(* CODESYS project wago_aws_iot_example_v0.2.01.ecp

Project tree, tasks and I/O mapping:
  PFC200_CS_2ETH_RS : 750-8202 PFC200 2ETH RS, WAGO, order no. 0750-8202, version 5.11.1.16
    application Application
      libraries: 
      task PLC_Task (cyclic, interval t#10ms, priority 14) calls PLC_PRG
      task VISU_TASK (cyclic, interval 100 ms, priority 15) calls VisuElems.Visu_Prg
      visualisation Visualization
      function block UPDATE_AWS_IOT_THING_SHADOW [ST]: PUB_STRING
      program PLC_PRG [ST]
      visualisation Shadow_Attribute_Visu
      image pool ImagePool
      function block GET_AWS_IOT_THING_SHADOW [ST]: CURL_STRING
      function funC_TO_F [ST]
    DeviceAdapter
    Kbus : Kbus, WAGO, version 1.4.0.2
        unmapped channels: K-BUS diagnostics
      _4_AI_4_20mA_s_e_1 : 0750-0455, WAGO, order no. 0750-0455, version 0.0.0.12
          settings: K-BUS Module slot index = 1
          unmapped channels: _IW 1, _IW 2, _IW 3, _IW 4
        DeviceAdapter
      _2_AO_4_20mA_1 : 0750-0554, WAGO, order no. 0750-0554, version 0.0.0.9
          settings: K-BUS Module slot index = 2
          output Application.PLC_PRG.wOutputSignal1 : WORD  // _QW 1
          unmapped channels: _QW 2
        DeviceAdapter
      _2_AI_Thermocouple_T_Diag : 0750-0469/0000-0002, WAGO, order no. 0750-0469/0000-0002, version 0.0.0.9
          settings: K-BUS Module slot index = 3
          input  Application.PLC_PRG.wTcInputRaw1 : INT  // _IINT 1
          unmapped channels: _IINT 2
        DeviceAdapter
    MODBUS
      MODBUS : MODBUS, WAGO, order no. n/a, version 1.1.1.15
    Serial
      COM1 : COM1, WAGO, version 0.0.0.19
  libraries: SysProcess, 3.5.7.0 (System); WagoSysString, 1.6.0.0 (WAGO); WagoAppFileDir, 1.6.1.0 (WAGO); VisuSymbols, 3.5.10.0 (System); WagoVisuIcons, 1.0.0.8 (WAGO)
  5ce3da45-db07-42e7-a21c-a00fff4ed8f6|Z:\Dropbox\Demos\e!Cockpit\AWS\AWS IoT Thing Demo\cloud-service-types.png
  text list GlobalTextList
  data type typIOT_THING_SHADOW
  5ce3da45-db07-42e7-a21c-a00fff4ed8f6|Z:\Dropbox\Demos\e!Cockpit\AWS\AWS IoT Thing Demo\aws-iot.jpg
  5ce3da45-db07-42e7-a21c-a00fff4ed8f6|Z:\Dropbox\Demos\e!Cockpit\AWS\AWS IoT Thing Demo\cloud_circuit_h256.png
  5ce3da45-db07-42e7-a21c-a00fff4ed8f6|Z:\Dropbox\Demos\e!Cockpit\AWS\AWS IoT Thing Demo\icon-cloud-service.jpg
  5ce3da45-db07-42e7-a21c-a00fff4ed8f6|Z:\Dropbox\Demos\e!Cockpit\AWS\AWS IoT Thing Demo\deck_compute_chip_300_1.png
  5ce3da45-db07-42e7-a21c-a00fff4ed8f6|Z:\Dropbox\Demos\e!Cockpit\AWS\AWS IoT Thing Demo\aws-iot-product.png
  5ce3da45-db07-42e7-a21c-a00fff4ed8f6|Z:\Dropbox\Demos\e!Cockpit\AWS\AWS IoT Thing Demo\WAGO_Logo_v1.png
*)

// typIOT_THING_SHADOW
TYPE typIOT_THING_SHADOW :
STRUCT
		sLabel	: STRING;
		sValue	: STRING;
END_STRUCT
END_TYPE

// PFC200_CS_2ETH_RS/Application/PLC_PRG
PROGRAM PLC_PRG
VAR
	fbAwsGetShadow			: GET_AWS_IOT_THING_SHADOW;
	fbAwsPutShadow			: UPDATE_AWS_IOT_THING_SHADOW;
	
	tonGetThingShadow		: TON;
	
	atypShadowAttributesIn	: ARRAY[1..1] OF typIOT_THING_SHADOW;
	atypShadowAttributesOut	: ARRAY[1..3] OF typIOT_THING_SHADOW;
	
	sAwsIotThingName		: STRING := 'WAGO_MSQ';
	sAwsRootCaPath			: STRING := '/etc/mosquitto/certs/rootCA.pem';
	sAwsCertPath			: STRING := '/etc/mosquitto/certs/MY_THING.cert.pem';
	sAwsKeyPath				: STRING := '/etc/mosquitto/certs/MY_THING.private.key';
	sAwsEndpoint			: STRING := '123456.iot.us-west-2.amazonaws.com';  
	sAwsShadowTopic			: STRING := '$$aws/things/MY_THING/shadow/update';
	
	xGetThingShadow			: BOOL;
	xPutThingShadow			: BOOL;
	xSyncAwsIotThingShadow	: BOOL;
	xIncrementShadow		: BOOL;
	
	wOutputSignal1			: WORD;
	wTcInputRaw1			: WORD;
	i						: INT;
	xTest					: BOOL := TRUE;
END_VAR

fbAwsGetShadow(
	xExecute:= xGetThingShadow, 
	Shadow_Attributes:= atypShadowAttributesIn, 
	sThingName:= sAwsIotThingName, 
	sRootCaPath:= sAwsRootCaPath, 
	sCertPath:= sAwsCertPath, 
	sKeyPath:= sAwsKeyPath, 
	sEndpoint:= sAwsEndpoint);
	
fbAwsPutShadow(
	xExecute:= xPutThingShadow, 
	Shadow_Attributes:= atypShadowAttributesOut, 
	sRootCaPath:= sAwsRootCaPath, 
	sCertPath:= sAwsCertPath, 
	sKeyPath:= sAwsKeyPath, 
	sEndpoint:= sAwsEndpoint, 
	sTopic:= sAwsShadowTopic);
	
IF xSyncAwsIotThingShadow THEN
	atypShadowAttributesOut[1] := atypShadowAttributesIn[1];
	xSyncAwsIotThingShadow := FALSE;
END_IF

IF NOT xTest THEN
	tonGetThingShadow(IN:= NOT xGetThingShadow, PT:= T#5S);
	IF tonGetThingShadow.Q THEN
		xGetThingShadow := TRUE;
		atypShadowAttributesOut[1] := atypShadowAttributesIn[1];
		xPutThingShadow := TRUE;
	END_IF
END_IF

wOutputSignal1 := STRING_TO_WORD(atypShadowAttributesIn[1].sValue);

atypShadowAttributesOut[2].sLabel := 'TempF';
atypShadowAttributesOut[2].sValue := REAL_TO_STRING(funC_TO_F(wTcInputRaw1));
atypShadowAttributesOut[3].sLabel := 'TempC';
atypShadowAttributesOut[3].sValue := WORD_TO_STRING(wTcInputRaw1 / 10);

END_PROGRAM

// PFC200_CS_2ETH_RS/Application/funC_TO_F
FUNCTION funC_TO_F : REAL
VAR_INPUT
	wTcRaw		: WORD;
END_VAR
VAR
	rTempHold	: REAL;
END_VAR

rTempHold := WORD_TO_REAL(wTcRaw / 10);
rTempHold := (rTempHold * 1.8) + 32;

funC_TO_F := rTempHold;

END_FUNCTION

// PFC200_CS_2ETH_RS/Application/GET_AWS_IOT_THING_SHADOW
FUNCTION_BLOCK GET_AWS_IOT_THING_SHADOW	
VAR_IN_OUT
	xExecute: BOOL;
	Shadow_Attributes	: ARRAY[*] OF typIOT_THING_SHADOW;
END_VAR
VAR_INPUT
	sThingName			: STRING;
	sRootCaPath			: STRING;
	sCertPath			: STRING;
	sKeyPath			: STRING;
	sEndpoint			: STRING;
END_VAR
VAR_OUTPUT
	//diTest				: DINT;
END_VAR
VAR
	sQueryBashScript	: STRING(255);
	sBashResponse: STRING;
	ptBashRslt: RTS_IEC_RESULT;
	diFileStatus: DINT;
	fbReadShadowFile: FbReadWholeFile_cpt;
	oReadFileStatus: FbResult;
	xReadFileTrig: BOOL;
	xREadFileError: BOOL;
	xREadFileBusy: BOOL;
	abFileData		: ARRAY[1..10000] OF BYTE;
	udiReadFileSize: UDINT := 10000;
	udiReadRxNumOfBytes: UDINT;
	xReadFileEndReached: BOOL;
	xConvertToTyp: BOOL;
	b: UDINT;
	xByteIsChar: BOOL;
	iCurlIndex: INT;
	xOnLabel: BOOL;
	xOnValue: BOOL;
	iWriteIndex: INT;
	sCurrentValueString: STRING;
	sCurrentLabelString: STRING;
	ub: DINT;
END_VAR

ub:=UPPER_BOUND (Shadow_Attributes,1);

IF xExecute THEN
	sQueryBashScript := CURL_STRING(
							sThingName:= sThingName, 
							sRootCaPath:= sRootCaPath, 
							sCertPath:= sCertPath, 
							sKeyPath:= sKeyPath, 
							sEndPoint:= sEndpoint);
	diFileStatus := SysProcessExecuteCommand2(pszCommand:= sQueryBashScript, pszStdOut:= sBashResponse, udiStdOutLen:= 255, pResult:= ptBashRslt);
	
	//diTest := diFileStatus;
	IF (diFileStatus <> 0) AND NOT xReadFileEndReached THEN
		xReadFileTrig := TRUE;
		fbReadShadowFile(
			oStatus=> oReadFileStatus, 
			xTrigger:= xReadFileTrig, 
			xError=> xREadFileError, 
			xBusy=> xREadFileBusy, 
			sName:= '/root/.rcv_shadow.json', 
			pRxBuffer:= ADR(abFileData), 
			udiRxBufferSize:= udiReadFileSize, 
			udiRxNBytes=> udiReadRxNumOfBytes, 
			xEofReached=> xReadFileEndReached);
		FOR b := 1 TO udiReadRxNumOfBytes DO
				//checks to see if the byte is an alpha-numeric
				IF 	((abFileData[b] >= 48) AND abFileData[b] <= 57) 	OR
					((abFileData[b] >= 65) AND abFileData[b] <= 90) 	OR
					((abFileData[b] >= 97) AND abFileData[b] <= 122) 	THEN
					xByteIsChar := TRUE;
				ELSE
					xByteIsChar := FALSE;
				END_IF
				
				// curly braces
				IF (abFileData[b] = 123) THEN
					iCurlIndex := iCurlIndex + 1;
				END_IF
				
				// if this is a new scan or the byte is a comma
				IF ((iCurlIndex = 3) AND (abFileData[b] = 123))  OR (abFileData[b] = 44) AND NOT xOnLabel THEN
					xOnLabel := TRUE;
					xOnValue := FALSE;
					Shadow_Attributes[iWriteIndex].sLabel:= sCurrentLabelString;
					Shadow_Attributes[iWriteIndex].sValue:= sCurrentValueString;
					sCurrentLabelString := '';
					sCurrentValueString := '';
					iWriteIndex := iWriteIndex + 1;
					
				//looks for a colon
				ELSIF (abFileData[b] = 58) THEN
					xOnLabel := FALSE;
					xOnValue := TRUE;
				END_IF
				
				IF xByteIsChar THEN
					IF xOnLabel THEN
						sCurrentLabelString := CONCAT(sCurrentLabelString, ASCIIBYTE_TO_STRING(abFileData[b]));
					ELSIF xOnValue THEN
						sCurrentValueString := CONCAT(sCurrentValueString, ASCIIBYTE_TO_STRING(abFileData[b]));
					END_IF
				END_IF

			IF iWriteIndex > ub THEN		
				// reseting variabel values here
				xReadFileEndReached := FALSE;
				xREadFileBusy := FALSE;
				xReadFileTrig := FALSE;
				xOnLabel := FALSE;
				xOnValue := FALSE;
				iCurlIndex := 0;
				iWriteIndex := 0;
				xExecute := FALSE;
				RETURN;
			END_IF
		END_FOR
	END_IF
END_IF

METHOD INTERNAL CURL_STRING : STRING(255)
VAR_INPUT
	sThingName	: STRING;
	sRootCaPath	: STRING;
	sCertPath	: STRING;
	sKeyPath	: STRING;
	sEndPoint	: STRING;
END_VAR

VAR
	sHoldString: STRING(255);
END_VAR
//mosquitto_pub --cafile $1 --cert $2 --key $3 -h $4 -p 8883 -q 1 -d -t $5 -f $6
//sh .rcv_shadow.sh /etc/mosquitto/certs/rootCA.pem /etc/mosquitto/certs/WAGO_MSQ.cert.pem /etc/mosquitto/certs/WAGO_MSQ.private.key  https://a149vimaq58p1y.iot.us-west-2.amazonaws.com:8443/things/WAGO_MSQ/shadow
//https://a149vimaq58p1y.iot.us-west-2.amazonaws.com:8443/things/WAGO_MSQ/shadow
sHoldString := 'sh /root/.rcv_shadow.sh ';
sHoldString := CONCAT(sHoldString, sRootCaPath);
sHoldString := CONCAT(sHoldString, ' ');
sHoldString := CONCAT(sHoldString, sCertPath);
sHoldString := CONCAT(sHoldString, ' ');
sHoldString := CONCAT(sHoldString, sKeyPath);
sHoldString := CONCAT(sHoldString, ' ');
sHoldString := CONCAT(sHoldString, sEndpoint);
sHoldString := CONCAT(sHoldString, ':8443/things/');
sHoldString := CONCAT(sHoldString, sThingName);
sHoldString := CONCAT(sHoldString, '/shadow');

CURL_STRING := sHoldString;
END_METHOD

END_FUNCTION_BLOCK

// PFC200_CS_2ETH_RS/Application/UPDATE_AWS_IOT_THING_SHADOW
FUNCTION_BLOCK UPDATE_AWS_IOT_THING_SHADOW
VAR_IN_OUT
	xExecute: BOOL;	// trigger to send the data to the AWS IoT Thing Shadow
	Shadow_Attributes	: ARRAY[*] OF typIOT_THING_SHADOW;
END_VAR
VAR_INPUT
	sRootCaPath			: STRING;
	sCertPath			: STRING;
	sKeyPath			: STRING;
	sEndpoint			: STRING;
	sTopic				: STRING;
END_VAR
VAR
	fbWriteFile			: FbWriteWholeFile_cpt;
	ub					: DINT;
	lb					: DINT;
	i					: DINT;
	sBaseString			: STRING(22) := '{"state":{"reported":{ ';
	sAttributeString	: STRING;
	aWriteBytes			: ARRAY[1..10000] OF BYTE;
	aHoldBytes			: ARRAY[1..80] OF BYTE;
	ptString 			: POINTER TO BYTE;
	l					: INT;
	diSizeOfString		: DINT;
	index				: INT;
	x: INT;
	sTestString: STRING(255);
	xWriteFile: BOOL;
	oWriteFileStatus: FbResult;
	xWriteFileTrig: BOOL;
	xWriteFileError: BOOL;
	xWriteFileBusy: BOOL;
	sWriteFileName: STRING := '/root/.send_shadow.json';
	sPublishBashScript: STRING(255);
	rtsSendResult: RTS_IEC_RESULT;
	sReturnResponse: STRING(255);
END_VAR

ub:=UPPER_BOUND (Shadow_Attributes,1);
lb:=LOWER_BOUND (Shadow_Attributes,1);

IF xExecute THEN
	index := 0;
	//begin building the array
	ptString := ADR(sBaseString);
	FOR l := 1 TO len(sBaseString) DO
		aWriteBytes[l] := ptString^;
		ptString := ptString + 1;
	END_FOR	
	ptString := 0;
	index := index + len(sBaseString);
	// write JSON header
	FOR i := lb TO ub DO /// loop through each atrribute / value
		sAttributeString := '"';
		sAttributeString := CONCAT(sAttributeString, Shadow_Attributes[i].sLabel);
		sAttributeString := CONCAT(sAttributeString, '": "');
		sAttributeString := CONCAT(sAttributeString, Shadow_Attributes[i].sValue);
		sAttributeString := CONCAT(sAttributeString, '"');
		IF (i < ub) THEN
			sAttributeString := CONCAT(sAttributeString, ',');
		ELSIF i = ub THEN
			sAttributeString := CONCAT(sAttributeString, '}}}');
		END_IF
		diSizeOfString := LEN(sAttributeString);
		ptString := ADR(sAttributeString);
		FOR l := 1 TO len(sAttributeString) DO
			aHoldBytes[l] := ptString^;
			ptString := ptString + 1;
			aWriteBytes[l + index] := aHoldBytes[l]; 
		END_FOR
		
		index := index + len(sAttributeString);
		
		IF i = ub THEN
			xWriteFileTrig := TRUE;
		END_IF
	END_FOR

// write the file
	fbWriteFile(
		oStatus=> oWriteFileStatus, 
		xTrigger:= xWriteFileTrig, 
		xError=> xWriteFileError, 
		xBusy=> xWriteFileBusy, 
		sName:= sWriteFileName, 
		pTxBuffer:= ADR(aWriteBytes), 
		udiTxNBytes:= index);
		
		IF NOT xWriteFileTrig THEN
			sPublishBashScript := PUB_STRING(
										sRootCaPath:= sRootCaPath, 
										sCertPath:= sCertPath, 
										sKeyPath:= sKeyPath, 
										sEndPoint:= sEndpoint, 
										sTopic:= sTopic);
			SysProcessExecuteCommand2(pszCommand:= sPublishBashScript, pszStdOut:= sReturnResponse, udiStdOutLen:= 255, pResult:= rtsSendResult);
			xExecute := FALSE;
		END_IF
END_IF

METHOD INTERNAL PUB_STRING : STRING(255)
VAR_INPUT
	sRootCaPath	: STRING;
	sCertPath	: STRING;
	sKeyPath	: STRING;
	sEndPoint	: STRING;
	sTopic		: STRING;
END_VAR

VAR
	sHoldString: STRING(255);
END_VAR
//mosquitto_pub --cafile $1 --cert $2 --key $3 -h $4 -p 8883 -q 1 -d -t $5 -f $6
sHoldString := 'sh /root/.send_shadow.sh ';
sHoldString := CONCAT(sHoldString, sRootCaPath);
sHoldString := CONCAT(sHoldString, ' ');
sHoldString := CONCAT(sHoldString, sCertPath);
sHoldString := CONCAT(sHoldString, ' ');
sHoldString := CONCAT(sHoldString, sKeyPath);
sHoldString := CONCAT(sHoldString, ' ');
sHoldString := CONCAT(sHoldString, sEndPoint);
sHoldString := CONCAT(sHoldString, ' $'');
sHoldString := CONCAT(sHoldString, sTopic);
sHoldString := CONCAT(sHoldString, '$' /root/.send_shadow.json');

PUB_STRING := sHoldString;
END_METHOD

END_FUNCTION_BLOCK

// PFC200_CS_2ETH_RS/Application/Visualization
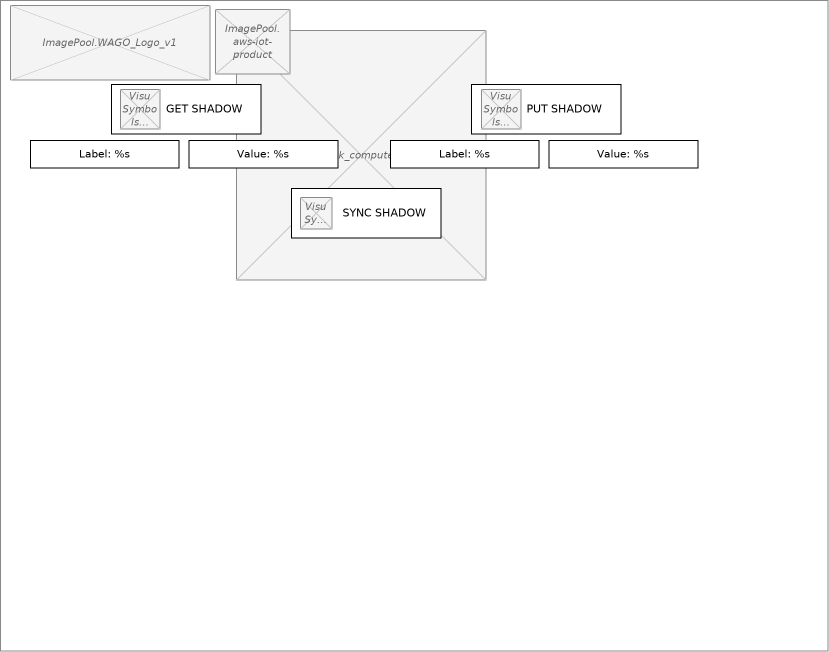
VISUALIZATION Visualization  // 829x652
    Rectangle (0,0 827x650)
    Image (236,30 250x250), image: ImagePool.deck_compute_chip_300_1
    Image (215,9 75x65), image: ImagePool.aws-iot-product
    Frame (30,140 310x30)
        shows Shadow_Attribute_Visu(typSA := PLC_PRG.atypShadowAttributesIn[1])
    Frame (390,140 310x30)
        shows Shadow_Attribute_Visu(typSA := PLC_PRG.atypShadowAttributesOut[1])
    Group (111,84 150x50)
        toggle PLC_PRG.xGetThingShadow
        RoundedRectangle (0,0 150x50)
        Image (9,5 40x40), image: VisuSymbols.Symbols.ArrowBoldDown
        Rectangle (37,8 113x34), "GET SHADOW"
    Group (471,84 150x50)
        toggle PLC_PRG.xPutThingShadow
        RoundedRectangle (0,0 150x50)
        Rectangle (37,8 113x34), "PUT SHADOW"
        Image (10,5 40x40), image: VisuSymbols.Symbols.ArrowBoldUp
    Image (10,5 200x75), image: ImagePool.WAGO_Logo_v1
    Group (291,188 150x50)
        toggle PLC_PRG.xSyncAwsIotThingShadow
        RoundedRectangle (0,0 150x50)
        Rectangle (37,8 113x34), "SYNC SHADOW"
        Image (9,9 32x32), image: VisuSymbols.Symbols.ArrowRoundLeftBottom
END_VISUALIZATION

// PFC200_CS_2ETH_RS/Application/Shadow_Attribute_Visu
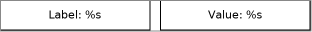
VISUALIZATION Shadow_Attribute_Visu  // 312x32
VAR_IN_OUT
	typSA	: typIOT_THING_SHADOW;
END_VAR
    Rectangle (0,0 150x30), "Label: %s", text variable: typSA.sLabel
    Rectangle (160,0 150x30), "Value: %s", text variable: typSA.sValue
        OnMouseDown: write the text variable via Edit
END_VISUALIZATION
